TYPE ST_Settings :
STRUCT
	iSP_WaterFillingMaxTime			:DINT;
END_STRUCT
END_TYPE

(* stored: Version 1.1.0.1, ProductVersion 3.1.4024.12
   DUT ST_Settings: Id {a12d9e13-6037-4b3c-8119-fd19efc51606} *)
